// TIA Portal project "Motor_Control_System_V1" (V17)

(* hardware
DEVICE "S7-1200 station_1"  S7-1200 Station
   slot 0: "Rack_0"  S7-1200 Rack  Rack  V1.0
   slot 1: "PLC_1"  CPU 1214C DC/DC/DC  6ES7 214-1AG40-0XB0  V4.5
DEVICE "HMI_1"  KTP700 Basic PN
   slot 0: "HMI_1"  KTP700 Basic PN  6AV2 123-2GB03-0AX0  17.0.0.0
   slot 1: "HMI_RT_1"  KTP700 Basic PN  6AV2 123-2GB03-0AX0  17.0.0.0
   slot 5: "HMI_1.IE_CP_1"  PROFINET Interface  17.0.0.0
      slot 1: "PROFINET Interface_1"  PROFINET Interface
         slot 1: "Port_1"  Port
*)

// ===== PLC "PLC_1"  CPU 1214C DC/DC/DC =====

VAR_GLOBAL   // PLC tag table "Physical_IO"
   "Start_Button" AT %I0.0 : Bool;   // 启动按钮
   "Stop_Button" AT %I0.1 : Bool;   // 停止按钮
   "Emergency_OK" AT %I0.2 : Bool;   // 急停按钮状态，1正常，0急停
   "Overload_OK" AT %I0.3 : Bool;   // 热继电器状态，1正常，0过载
   "Motor_Feedback" AT %I0.4 : Bool;   // 接触器辅助触点反馈
   "Motor_Contactor" AT %Q0.0 : Bool;   // 电机主接触器线圈
END_VAR

DATA_BLOCK "DB_Motor"   // DB1
{ S7_Optimized_Access := 'TRUE' }
VERSION : 0.1
   VAR
      Command : Struct   // 控制命令
         Start : Bool;   // 启动命令
         Stop : Bool;   // 停止命令
         Reset : Bool;   // 故障复位命令
      END_STRUCT;
      Status : Struct   // 运行状态
         Running : Bool;   // 电机是否在运行状态
         Ready : Bool;   // 设备允许运行状态
         Fault : Bool;   // 电机故障状态
         Feedback_OK : Bool;   // 电机反馈正常
         Feedback_Fault : Bool;   // 电机反馈故障
         State : Int;   // 电机状态 0停止 1准备就绪 2运行中 3故障
      END_STRUCT;
      HMI : Struct   // HMI控制命令
         Start_CMD : Bool;   // 触摸屏启动按钮
         Stop_CMD : Bool;   // 触摸屏停止按钮
      END_STRUCT;
   END_VAR
BEGIN
END_DATA_BLOCK

DATA_BLOCK "DB_CSharp"   // DB3
{ S7_Optimized_Access := 'FALSE' }
VERSION : 0.1
   VAR
      Start_CMD : Bool;
      Stop_CMD : Bool;
      Ready : Bool;
      Running : Bool;
      Fault : Bool;
      Feedback_Fault : Bool;
      Reset_CMD : Bool;
      State : Int;
      Emergency_OK : Bool;
      Overload_OK : Bool;
      Motor_Feedback : Bool;
   END_VAR
BEGIN
END_DATA_BLOCK

// folder: System blocks/Program resources

DATA_BLOCK "DB_Motor_Feedback_Timer"   // DB2
{ S7_Optimized_Access := 'TRUE' }
AUTHOR : Simatic
FAMILY : IEC
NAME : IEC_TMR
VERSION : 1.0
// stored: InstanceOfName IEC_TIMER
"IEC_TIMER"
BEGIN
END_DATA_BLOCK

// folder: (top level)

FUNCTION "FC_Motor_Control" : Void   // FC10, LAD
TITLE = 电机控制功能
{ S7_Optimized_Access := 'TRUE' }
VERSION : 0.1
BEGIN

REGION Network 1: 设备运行许可判断
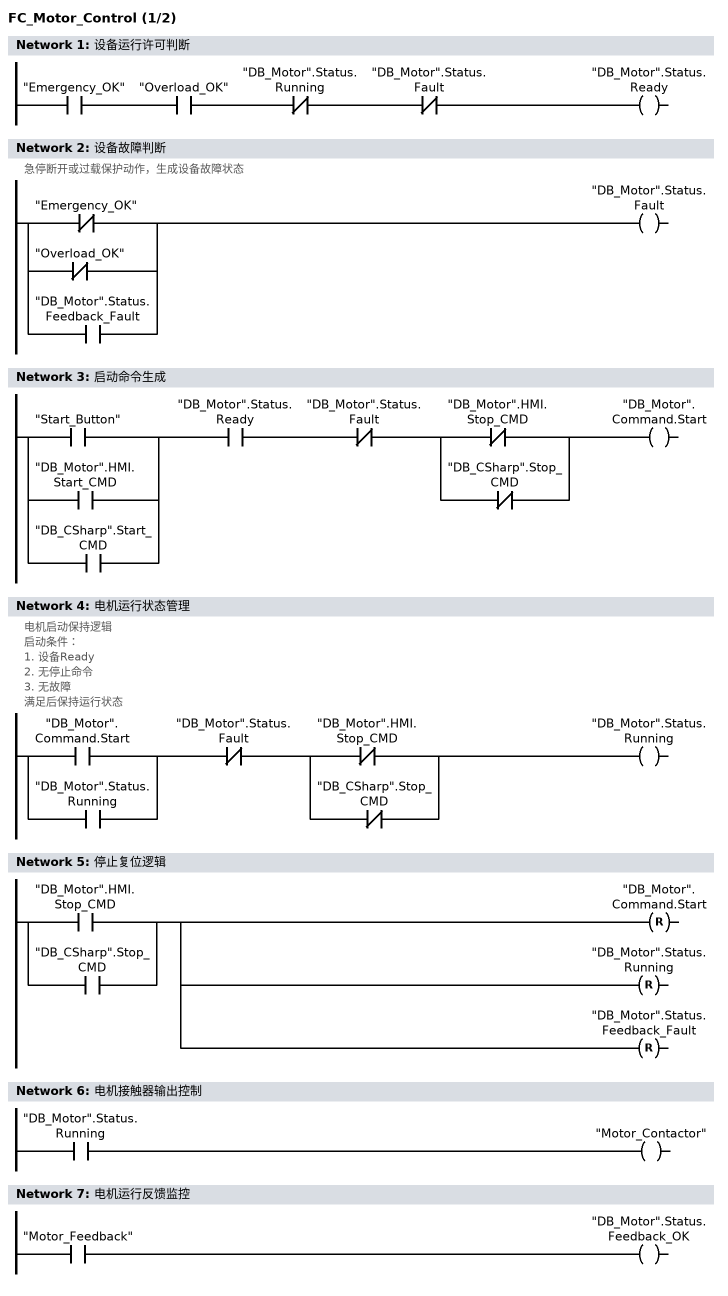
   RUNG wire#powerrail
      Contact( "Emergency_OK" )
      Contact( "Overload_OK" )
      I_Contact( "DB_Motor".Status.Running )
      I_Contact( "DB_Motor".Status.Fault )
      Coil( "DB_Motor".Status.Ready )
   END_RUNG
   // the same network as SCL:
   "DB_Motor".Status.Ready := "Emergency_OK" AND "Overload_OK" AND NOT "DB_Motor".Status.Running AND NOT "DB_Motor".Status.Fault;
END_REGION

REGION Network 2: 设备故障判断
   // 急停断开或过载保护动作，生成设备故障状态
   RUNG wire#powerrail
      I_Contact( "Emergency_OK" )
      wire#w1
      Coil( "DB_Motor".Status.Fault )
   END_RUNG
   RUNG wire#powerrail
      I_Contact( "Overload_OK" )
   END_RUNG wire#w1
   RUNG wire#powerrail
      Contact( "DB_Motor".Status.Feedback_Fault )
   END_RUNG wire#w1
   // the same network as SCL:
   "DB_Motor".Status.Fault := NOT "Emergency_OK" OR NOT "Overload_OK" OR "DB_Motor".Status.Feedback_Fault;
END_REGION

REGION Network 3: 启动命令生成
   RUNG wire#powerrail
      Contact( "Start_Button" )
      wire#w1
      Contact( "DB_Motor".Status.Ready )
      I_Contact( "DB_Motor".Status.Fault )
      wire#w2
      I_Contact( "DB_Motor".HMI.Stop_CMD )
      wire#w3
      Coil( "DB_Motor".Command.Start )
   END_RUNG
   RUNG wire#powerrail
      Contact( "DB_Motor".HMI.Start_CMD )
   END_RUNG wire#w1
   RUNG wire#powerrail
      Contact( "DB_CSharp".Start_CMD )
   END_RUNG wire#w1
   RUNG wire#w2
      I_Contact( "DB_CSharp".Stop_CMD )
   END_RUNG wire#w3
   // the same network as SCL:
   "DB_Motor".Command.Start := ("Start_Button" OR "DB_Motor".HMI.Start_CMD OR "DB_CSharp".Start_CMD) AND "DB_Motor".Status.Ready AND NOT "DB_Motor".Status.Fault AND (NOT "DB_Motor".HMI.Stop_CMD OR NOT "DB_CSharp".Stop_CMD);
END_REGION

REGION Network 4: 电机运行状态管理
   // 电机启动保持逻辑
   // 
   // 
   // 启动条件：
   // 
   // 1. 设备Ready 
   // 
   // 2. 无停止命令
   // 
   // 3. 无故障
   // 
   // 
   // 满足后保持运行状态
   RUNG wire#powerrail
      Contact( "DB_Motor".Command.Start )
      wire#w1
      I_Contact( "DB_Motor".Status.Fault )
      wire#w2
      I_Contact( "DB_Motor".HMI.Stop_CMD )
      wire#w3
      Coil( "DB_Motor".Status.Running )
   END_RUNG
   RUNG wire#powerrail
      Contact( "DB_Motor".Status.Running )
   END_RUNG wire#w1
   RUNG wire#w2
      I_Contact( "DB_CSharp".Stop_CMD )
   END_RUNG wire#w3
   // the same network as SCL:
   "DB_Motor".Status.Running := ("DB_Motor".Command.Start OR "DB_Motor".Status.Running) AND NOT "DB_Motor".Status.Fault AND (NOT "DB_Motor".HMI.Stop_CMD OR NOT "DB_CSharp".Stop_CMD);
END_REGION

REGION Network 5: 停止复位逻辑
   RUNG wire#powerrail
      Contact( "DB_Motor".HMI.Stop_CMD )
      wire#w1
      R_Coil( "DB_Motor".Command.Start )
   END_RUNG
   RUNG wire#powerrail
      Contact( "DB_CSharp".Stop_CMD )
   END_RUNG wire#w1
   RUNG wire#w1
      R_Coil( "DB_Motor".Status.Running )
   END_RUNG
   RUNG wire#w1
      R_Coil( "DB_Motor".Status.Feedback_Fault )
   END_RUNG
   // the same network as SCL:
   IF "DB_Motor".HMI.Stop_CMD OR "DB_CSharp".Stop_CMD THEN
       "DB_Motor".Command.Start := FALSE;
       "DB_Motor".Status.Running := FALSE;
       "DB_Motor".Status.Feedback_Fault := FALSE;
   END_IF;
END_REGION

REGION Network 6: 电机接触器输出控制
   RUNG wire#powerrail
      Contact( "DB_Motor".Status.Running )
      Coil( "Motor_Contactor" )
   END_RUNG
   // the same network as SCL:
   "Motor_Contactor" := "DB_Motor".Status.Running;
END_REGION

REGION Network 7: 电机运行反馈监控
   RUNG wire#powerrail
      Contact( "Motor_Feedback" )
      Coil( "DB_Motor".Status.Feedback_OK )
   END_RUNG
   // the same network as SCL:
   "DB_Motor".Status.Feedback_OK := "Motor_Feedback";
END_REGION

REGION Network 8: 电机反馈检测定时
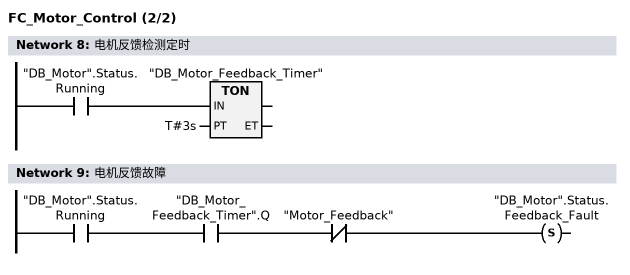
   "DB_Motor_Feedback_Timer".TON(IN := "DB_Motor".Status.Running, PT := T#3s);
END_REGION

REGION Network 9: 电机反馈故障
   RUNG wire#powerrail
      Contact( "DB_Motor".Status.Running )
      Contact( "DB_Motor_Feedback_Timer".Q )
      I_Contact( "Motor_Feedback" )
      S_Coil( "DB_Motor".Status.Feedback_Fault )
   END_RUNG
   // the same network as SCL:
   IF "DB_Motor".Status.Running AND "DB_Motor_Feedback_Timer".Q AND NOT "Motor_Feedback" THEN
       "DB_Motor".Status.Feedback_Fault := TRUE;
   END_IF;
END_REGION

REGION Network 10 (SCL): 电机状态汇总
   IF "DB_Motor".Status.Fault THEN
       "DB_Motor".Status.State := 3;
   ELSIF "DB_Motor".Status.Running THEN
       "DB_Motor".Status.State := 2;
   ELSIF "DB_Motor".Status.Ready THEN
       "DB_Motor".Status.State := 1;
   ELSE
       "DB_Motor".Status.State := 0;
   END_IF;
END_REGION

REGION Network 11 (SCL): C# 状态镜像
   // PLC → C#
   "DB_CSharp".Ready := "DB_Motor".Status.Ready;
   "DB_CSharp".Running := "DB_Motor".Status.Running;
   "DB_CSharp".Fault := "DB_Motor".Status.Fault;
   "DB_CSharp".Feedback_Fault := "DB_Motor".Status.Feedback_Fault;
   "DB_CSharp".State := "DB_Motor".Status.State;

   "DB_CSharp".Emergency_OK := "Emergency_OK";
   "DB_CSharp".Overload_OK := "Overload_OK";
   "DB_CSharp".Motor_Feedback := "Motor_Feedback";
END_REGION
END_FUNCTION

ORGANIZATION_BLOCK "Main"   // OB1, LAD, ProgramCycle
TITLE = "Main Program Sweep (Cycle)" / 主程序
{ S7_Optimized_Access := 'TRUE' }
VERSION : 0.1
   VAR_INPUT
      Initial_Call : Bool;   // Initial call of this OB
      Remanence : Bool;   // =True, if remanent data are available
   END_VAR
BEGIN

REGION Network 1: 电机控制功能调用
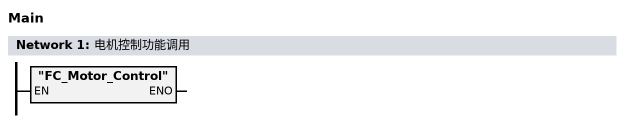
   RUNG wire#powerrail
      "FC_Motor_Control"()
   END_RUNG
   // the same network as SCL:
   "FC_Motor_Control"();
END_REGION
END_ORGANIZATION_BLOCK

(* ===== HMI "HMI_RT_1" =====
system functions are stored by id; their names below are inferred from use
connection "HMI_连接_1": ETHERNET, SMART_S7_1200_OMS

HMI tags "默认变量表"
   "Tag_ScreenNumber" : UInt, internal
   "DB_Motor_Status_Running" : Bool = PLC DB_Motor.Status.Running, 1 s
   "DB_Motor_Status_Ready" : Bool = PLC DB_Motor.Status.Ready, 1 s
   "DB_Motor_Status_Fault" : Bool = PLC DB_Motor.Status.Fault, 1 s
   "Emergency_OK" : Bool = PLC Emergency_OK AT %I0.2, 1 s
   "Overload_OK" : Bool = PLC Overload_OK AT %I0.3, 1 s

HMI tags "变量表_1"
   "HMI_Start_CMD" : Bool = PLC DB_Motor.HMI.Start_CMD, 1 s
   "HMI_Stop_CMD" : Bool = PLC DB_Motor.HMI.Stop_CMD AT %DB1.DBX0.0, 1 s
   "HMI_Motor_State" : Int = PLC DB_Motor.Status.State AT %DB1.DBX0.0, 1 s

text list "Motor_State_List": 0 '停止'; 1 '准备就绪'; 2 '运行中'; 3 '故障'

Template "模板_1" 800x480
   Button "退出" at 714,429 size 71x50; TextOff '退出'; PictureOff "ExitRuntime_KTP700_Basic_PN_TR"; PictureOn "ExitRuntime_KTP700_Basic_PN_TR"
      on Release: StopRuntime(0)
   Button "Template_Button" at 614,429 size 71x50; TextOff 'Text'
   Button "Template_Button_1" at 514,429 size 71x50; TextOff 'Text'
   Button "Template_Button_2" at 414,429 size 71x50; TextOff 'Text'
   Button "Template_Button_3" at 314,429 size 71x50; TextOff 'Text'
   Button "Template_Button_4" at 214,429 size 71x50; TextOff 'Text'
   Button "报警" at 114,429 size 71x50; TextOff '报警'; PictureOff "AlarmDisplay_KTP700_Basic_PN_TR"; PictureOn "AlarmDisplay_KTP700_Basic_PN_TR"
      on Release: function_ef3f5d25("报警窗口_Unacknowledged", -1)
   Button "起始画面" at 14,429 size 71x50; TextOff '起始画面'; PictureOff "NavigateHome_KTP700_Basic_PN_TR"; PictureOn "NavigateHome_KTP700_Basic_PN_TR"
      on Release: ActivateScreen("根画面", 0)
   DateTimeField "HmiScreenItemData" at 695,25 size 105x25
   DateTimeField "HmiScreenItemData_1" at 695,0 size 105x25
   GraphicView "Logo" at 0,0 size 91x51; Picture "HMI_1 的 Logo"

screen "根画面" 800x480, template "模板_1"
   on GenerateScreen: SetTag("Tag_ScreenNumber", 1)
   TextField "HmiScreenItemData" at 79,15 size 640x32; Text '电机控制系统'
   TextField "文本域_2" at 166,99 size 90x20; Text '运行状态灯'
   TextField "文本域_1" at 344,100 size 90x20; Text '准备状态灯'
   TextField "文本域_3" at 520,101 size 90x20; Text '故障状态灯'
   Circle "圆_1" at 138,93 size 28x28
      Appearance <- "DB_Motor_Status_Running"
   Circle "圆_2" at 316,94 size 28x28
      Appearance <- "DB_Motor_Status_Ready"
   Circle "圆_3" at 492,96 size 28x28
      Appearance <- "DB_Motor_Status_Fault"
   Button "按钮_1" at 198,184 size 120x45; TextOff '启动'
      on Press: SetBit("HMI_Start_CMD")
      on Release: ResetBit("HMI_Start_CMD")
   Button "按钮_2" at 390,184 size 120x45; TextOff '停止'
      on Press: SetBit("HMI_Stop_CMD")
      on Release: ResetBit("HMI_Stop_CMD")
   TextField "文本域_4" at 134,279 size 90x20; Text '设备状态：'
   TextField "文本域_8" at 134,319 size 90x20; Text '急停状态：'
   TextField "文本域_9" at 134,356 size 90x20; Text '过载状态：'
   TextField "文本域_10" at 221,319 size 39x20; Text '正常'
      Visibility <- "Emergency_OK"
   TextField "文本域_11" at 221,356 size 39x20; Text '正常'
      Visibility <- "Overload_OK"
   TextField "文本域_12" at 220,319 size 73x20; Text '急停触发'
      Visibility <- "Emergency_OK"
   TextField "文本域_13" at 222,355 size 39x20; Text '过载'
      Visibility <- "Overload_OK"
   SymbolicIOField "符号 I/O 域_1" at 222,272 size 129x32; TextOff '0'; TextOn '1'; TextList "Motor_State_List"
      ProcessValue <- "HMI_Motor_State"
*)